// Path identifier interface.
INTERFACE I_Path

// Full generated path including options.
PROPERTY Get : Str
GET
END_GET
END_PROPERTY

// TRUE when the path contains sSegment.
METHOD Has : BOOL
VAR_INPUT
	sSegment: Str; // Segment to find.
END_VAR
END_METHOD

// Full path length including options.
PROPERTY Length : USINT
GET
END_GET
END_PROPERTY

// Generated path without options.
PROPERTY Name : Str
GET
END_GET
END_PROPERTY

// Optional query-style path segment.
PROPERTY Option : Str
GET
END_GET
SET
END_SET
END_PROPERTY

END_INTERFACE

(* stored: Version 1.1.0.1
   Itf I_Path: Id {b955facb-7d92-45ed-9f56-bffab42f8eff}
   Property Get: Id {fe919d4f-04bf-47bd-952f-68f25ab34989}
   Get Get: Id {1eefc9f4-115f-48d5-9277-198342446fa8}
   Method Has: Id {b8393d0a-c05d-4bd2-96be-faa36956f3c3}
   Property Length: Id {6161492d-ccbd-4fab-931c-6a0a16cfbe97}
   Get Get: Id {75307abd-3222-476b-8b5e-8ccb26092503}
   Property Name: Id {1648e52e-030a-4aed-95b8-294b23471c90}
   Get Get: Id {c514d655-a1c7-43ca-957f-b0dc52f91241}
   Property Option: Id {c2c8963d-06eb-416b-a110-0e985fb960a6}
   Get Get: Id {d32ce12a-4979-49d2-8c44-8008d3b3eca5}
   Set Set: Id {ae001f47-64b0-45fc-bd00-108a840ea6c7} *)
